// TIA Portal V19 export
FUNCTION_BLOCK "CalledInPreInterpolator"   // FB154, LAD
AUTHOR : Siemens_FA_SUP
// stored: Access Published, MemoryReserve 100, Namespace Unit.Em2, SetENOAutomatically false
BEGIN

REGION Network 1
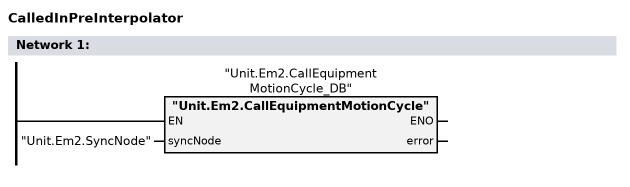
   RUNG wire#powerrail
      "Unit.Em2.CallEquipmentMotionCycle_DB"(syncNode := "Unit.Em2.SyncNode", error =>)
   END_RUNG
   // the same network as SCL:
   "Unit.Em2.CallEquipmentMotionCycle_DB"(syncNode := "Unit.Em2.SyncNode");   // "Unit.Em2.CallEquipmentMotionCycle"
END_REGION
END_FUNCTION_BLOCK
